PROGRAM master
VAR
END_VAR

END_PROGRAM

(* stored: Version 1.1.0.1, ProductVersion 3.1.4024.4
   POU master: Id {220e2799-3fee-4b6d-a227-2b1be6f3ade4}, SpecialFunc None *)
